// TIA Portal V17 export
// export: Created 2024-08-29T18:23:44.7165892Z, ExportSetting WithDefaults, DisplayName Totally Integrated Automation Portal, DisplayVersion V17 Update 7, DisplayName TIA Portal Openness, DisplayVersion V17 Update 7, DisplayName TIA Portal Version Control Interface, DisplayVersion V17, DisplayName SINAMICS Startdrive Advanced, DisplayVersion V17 SP2, DisplayName SINAMICS Startdrive G110M, G120, G120C, G120D, G120P, G115D, DisplayVersion V17 SP2, DisplayName SINAMICS Startdrive G130, G150, S120, S150, SINAMICS MV, S210, DisplayVersion V17 SP2, DisplayName STEP 7 Professional, DisplayVersion V17 Update 7, DisplayName STEP 7 Safety, DisplayVersion V17 Update 6, DisplayName WinCC Advanced / Unified PC, DisplayVersion V17 Update 7
DATA_BLOCK "labels"   // DB6
{ S7_Optimized_Access := 'TRUE' }
VERSION : 0.1
// stored: AutoNumber false, DBAccessibleFromOPCUA true, DBAccessibleFromWebserver true, IsOnlyStoredInLoadMemory false, IsRetainMemResEnabled false, IsWriteProtectedInAS false, MemoryReserve 100
   VAR RETAIN
      label1 : Array[0..32] of String[50];   // Etiqueta 1
      label2 : Array[0..32] of String[50];
      label3 : Array[0..32] of String[50];
      label4 : Array[0..32] of String[50];
      label5 : Array[0..32] of String[50];
      label6 : Array[0..32] of String[50];
      posLabel1 : Array[0..32] of Int;   // Posición de etiqueta 1
      posLabel2 : Array[0..32] of Int;
      posLabel3 : Array[0..32] of Int;
      posLabel4 : Array[0..32] of Int;
      posLabel5 : Array[0..32] of Int;
      posLabel6 : Array[0..32] of Int;
      text : Array[0..5] of String;   // Texto HMI de etiquetas
   END_VAR
   VAR
      done2 : Bool := FALSE;
      errorPort2 : Bool := FALSE;
      statusPort2 : Word := 16#7000;
      statusReset : Word := 16#7000;
   END_VAR
   VAR RETAIN
      doneReset : Bool := FALSE;
      scanner1 : Bool := TRUE;
      scanner2 : Bool := TRUE;
      scanner3 : Bool := TRUE;
      scanner4 : Bool := FALSE;
      scanner5 : Bool := FALSE;
   END_VAR
   VAR
      scanner6 : Bool := FALSE;
      scannerOn : Bool := TRUE;
      codeScanned : String := ' ';
      codeReceived : String := '';
      ndr : Bool := FALSE;
      error : Bool := FALSE;
      status : Word := 16#7002;
      lenght : UInt := 0;
      lablelBlock : Array[0..6] of Bool;
      nestScannerRead : String := ' ';
      readScanner : String := '03804073GO23548$R';
      extraction : Array[0..6] of String;
      previousBarcode : String := '';
   END_VAR
BEGIN
   label1[0..4] := '038';
   label1[5] := '1';
   label1[6..8] := '038';
   label1[9] := '202';
   label1[10..11] := '592';
   label1[12] := '202';
   label1[13] := '592';
   label1[14] := '202';
   label1[15..16] := '';
   label1[17] := '592';
   label1[18] := '202';
   label1[19] := '592';
   label1[20..32] := '';
   label2[0..1] := '4066654';
   label2[2] := '4066308';
   label2[3] := '4066654';
   label2[4] := '4066308';
   label2[5] := '2';
   label2[6..7] := '709';
   label2[8] := '706';
   label2[9] := '723';
   label2[10] := '724';
   label2[11] := '723';
   label2[12] := '724';
   label2[13] := '769';
   label2[14] := '768';
   label2[15..16] := '';
   label2[17..18] := '685';
   label2[19] := '163';
   label2[20..32] := '';
   label3[0..1] := '4066430';
   label3[2] := '4066646';
   label3[3] := '4066430';
   label3[4] := '4066646';
   label3[5] := '3';
   label3[6..7] := '708';
   label3[8] := '707';
   label3[9] := '718';
   label3[10] := '719';
   label3[11] := '718';
   label3[12..14] := '719';
   label3[15..16] := '';
   label3[17..18] := '680';
   label3[19] := '161';
   label3[20..32] := '';
   label4[0..32] := '';
   label5[0..32] := '';
   label6[0..32] := '';
   posLabel1[0..14] := 1;
   posLabel1[15..16] := 0;
   posLabel1[17..19] := 1;
   posLabel1[20..32] := 0;
   posLabel2[0..4] := 1;
   posLabel2[5] := 2;
   posLabel2[6..8] := 10;
   posLabel2[9..12] := 5;
   posLabel2[13..14] := 1;
   posLabel2[15..16] := 0;
   posLabel2[17..19] := 5;
   posLabel2[20..32] := 0;
   posLabel3[0..4] := 1;
   posLabel3[5] := 3;
   posLabel3[6..8] := 10;
   posLabel3[9..13] := 5;
   posLabel3[14] := 13;
   posLabel3[15..16] := 0;
   posLabel3[17..19] := 5;
   posLabel3[20..32] := 0;
   posLabel4[0..32] := 0;
   posLabel5[0..32] := 0;
   posLabel6[0..32] := 0;
   text[0] := '';
   text[1] := 'Motor';
   text[2] := 'Track Izq';
   text[3] := 'Track der';
   text[4..5] := '';
   lablelBlock[0] := FALSE;
   lablelBlock[1..3] := TRUE;
   lablelBlock[4..6] := FALSE;
   extraction[0] := '';
   extraction[1] := '038';
   extraction[2..3] := '0380407';
   extraction[4..6] := '';
END_DATA_BLOCK
